{attribute addProperty BoxType "EM7004-0000-0017"}
{attribute addProperty Id "Input_0BIT10.1251Input_1BIT10.1252Input_2BIT10.1253Input_3BIT10.1254Input_4BIT10.1255Input_5BIT10.1256Input_6BIT10.1257Input_7BIT10.1258Input_8BIT10.1259Input_9BIT10.12510Input_10BIT10.12511Input_11BIT10.12512Input_12BIT10.12513Input_13BIT10.12514Input_14BIT10.12515Input_15BIT10.12516"}
{attribute addProperty CRC "3496725889"}
{attribute addProperty SizeInBites "16"}
{attribute addProperty SizeInBytes "2"}
TYPE Input_D06BCD81 :
STRUCT
	{attribute addProperty Name "Input_0"}
	Input_0 : BIT;
	{attribute addProperty Name "Input_1"}
	Input_1 : BIT;
	{attribute addProperty Name "Input_2"}
	Input_2 : BIT;
	{attribute addProperty Name "Input_3"}
	Input_3 : BIT;
	{attribute addProperty Name "Input_4"}
	Input_4 : BIT;
	{attribute addProperty Name "Input_5"}
	Input_5 : BIT;
	{attribute addProperty Name "Input_6"}
	Input_6 : BIT;
	{attribute addProperty Name "Input_7"}
	Input_7 : BIT;
	{attribute addProperty Name "Input_8"}
	Input_8 : BIT;
	{attribute addProperty Name "Input_9"}
	Input_9 : BIT;
	{attribute addProperty Name "Input_10"}
	Input_10 : BIT;
	{attribute addProperty Name "Input_11"}
	Input_11 : BIT;
	{attribute addProperty Name "Input_12"}
	Input_12 : BIT;
	{attribute addProperty Name "Input_13"}
	Input_13 : BIT;
	{attribute addProperty Name "Input_14"}
	Input_14 : BIT;
	{attribute addProperty Name "Input_15"}
	Input_15 : BIT;
END_STRUCT
END_TYPE

(* stored: Version 1.2.0.0, ProductVersion 3.1.4024.9
   DUT Input_D06BCD81: Id {481aa5bc-4bd0-430a-9856-d07dd225db07} *)
